Fanuc TP program (LS listing): 12_from_to_points.ls

/PROG MOVE_SAFE_TO_PURGE_TO_HOME
/ATTR
OWNER = MNEDITOR;
COMMENT = "auto";
/MN
   1:  UFRAME_NUM=1 ;
   2:  UTOOL_NUM=1 ;
   3:  !move from safe travel point to purge station then return home ;
   4:  J PR[14:safe travel point] 100% FINE ;
   5:  L PR[16:purge station] 100mm/sec FINE ;
   6:  L PR[1:home] 100mm/sec FINE ;
/POS
/END
